// TIA Portal V16 export
// export: Created 2024-04-23T10:19:32.3047454Z, ExportSetting WithDefaults, DisplayName Totally Integrated Automation Portal, DisplayVersion V16 Update 5, DisplayName TIA Portal Version Control Interface, DisplayVersion V16 Update 2, DisplayName TIA Portal Openness, DisplayVersion V16 Update 5, DisplayName TIA Portal Teamcenter Gateway, DisplayVersion V16, DisplayName SINAMICS Startdrive Advanced, DisplayVersion V16, DisplayName SINAMICS Startdrive G130, G150, S120, S150, SINAMICS MV, S210, DisplayVersion V16, DisplayName SINAMICS Startdrive G110M, G120, G120C, G120D, G120P, DisplayVersion V16, DisplayName STEP 7 Professional, DisplayVersion V16 Update 5, DisplayName STEP 7 Safety, DisplayVersion V16, DisplayName WinCC UA Professional, DisplayVersion V16 Update 5
DATA_BLOCK "Calculo de Seno_DB"   // DB1
VERSION : 0.1
// stored: AutoNumber true, DBAccessibleFromOPCUA true, InstanceOfName Calculo de Seno, InstanceOfType FB
"Calculo de Seno"
   // VAR_OUTPUT
   //    SenOUT : Real;
   // END_VAR
   // VAR_IN_OUT
   //    SenIN : Real;
   // END_VAR
   // VAR
   //    Pulso1ms : Bool;
   //    AuxPulso1ms : Bool;
   //    AuxFlancoPulso4ms : Bool;
   //    Flanco4ms { ExternalAccessible := 'False'; ExternalVisible := 'False'; ExternalWritable := 'False'} : Bool;
   // END_VAR
BEGIN
END_DATA_BLOCK
